# EPICS substitutions: apps/caenHvApp/Db/subs/HVECAL5_SPARES.substitutions
#
#This file was autogenerated by mkHVEpics.C on: Wed Nov  2 16:01:55 2016
#Substitutions for crate: HVECAL5 SPARES
#
file "db/caenhv.db" {
        pattern { Cr,    CrName,         CrType, Sl,     Ch,    Sys,     Det,    Element,                CScode, pwonoff, v0set,  i0set,   trip,    rampup,  rampdn, svmax,   enable}
		{"10",	"HVECAL5",	"4527",	"09",	"00",	"HV",	"HVECAL5",	"SPARE_Sl09_Ch00",	"#C2314", "S2816", "S512", "S1280", "S2560", "S1024", "S768", "S3328", "S256"}
		{"10",	"HVECAL5",	"4527",	"09",	"01",	"HV",	"HVECAL5",	"SPARE_Sl09_Ch01",	"#C2314", "S2817", "S513", "S1281", "S2561", "S1025", "S769", "S3329", "S257"}
		{"10",	"HVECAL5",	"4527",	"09",	"02",	"HV",	"HVECAL5",	"SPARE_Sl09_Ch02",	"#C2314", "S2818", "S514", "S1282", "S2562", "S1026", "S770", "S3330", "S258"}
		{"10",	"HVECAL5",	"4527",	"09",	"03",	"HV",	"HVECAL5",	"SPARE_Sl09_Ch03",	"#C2314", "S2819", "S515", "S1283", "S2563", "S1027", "S771", "S3331", "S259"}
		{"10",	"HVECAL5",	"4527",	"09",	"04",	"HV",	"HVECAL5",	"SPARE_Sl09_Ch04",	"#C2314", "S2820", "S516", "S1284", "S2564", "S1028", "S772", "S3332", "S260"}
		{"10",	"HVECAL5",	"4527",	"09",	"05",	"HV",	"HVECAL5",	"SPARE_Sl09_Ch05",	"#C2314", "S2821", "S517", "S1285", "S2565", "S1029", "S773", "S3333", "S261"}
		{"10",	"HVECAL5",	"4527",	"09",	"06",	"HV",	"HVECAL5",	"SPARE_Sl09_Ch06",	"#C2314", "S2822", "S518", "S1286", "S2566", "S1030", "S774", "S3334", "S262"}
		{"10",	"HVECAL5",	"4527",	"09",	"07",	"HV",	"HVECAL5",	"SPARE_Sl09_Ch07",	"#C2314", "S2823", "S519", "S1287", "S2567", "S1031", "S775", "S3335", "S263"}
		{"10",	"HVECAL5",	"4527",	"09",	"08",	"HV",	"HVECAL5",	"SPARE_Sl09_Ch08",	"#C2314", "S2824", "S520", "S1288", "S2568", "S1032", "S776", "S3336", "S264"}
		{"10",	"HVECAL5",	"4527",	"09",	"09",	"HV",	"HVECAL5",	"SPARE_Sl09_Ch09",	"#C2314", "S2825", "S521", "S1289", "S2569", "S1033", "S777", "S3337", "S265"}
		{"10",	"HVECAL5",	"4527",	"09",	"10",	"HV",	"HVECAL5",	"SPARE_Sl09_Ch10",	"#C2314", "S2826", "S522", "S1290", "S2570", "S1034", "S778", "S3338", "S266"}
		{"10",	"HVECAL5",	"4527",	"09",	"11",	"HV",	"HVECAL5",	"SPARE_Sl09_Ch11",	"#C2314", "S2827", "S523", "S1291", "S2571", "S1035", "S779", "S3339", "S267"}
		{"10",	"HVECAL5",	"4527",	"09",	"12",	"HV",	"HVECAL5",	"SPARE_Sl09_Ch12",	"#C2314", "S2828", "S524", "S1292", "S2572", "S1036", "S780", "S3340", "S268"}
		{"10",	"HVECAL5",	"4527",	"09",	"13",	"HV",	"HVECAL5",	"SPARE_Sl09_Ch13",	"#C2314", "S2829", "S525", "S1293", "S2573", "S1037", "S781", "S3341", "S269"}
		{"10",	"HVECAL5",	"4527",	"09",	"14",	"HV",	"HVECAL5",	"SPARE_Sl09_Ch14",	"#C2314", "S2830", "S526", "S1294", "S2574", "S1038", "S782", "S3342", "S270"}
		{"10",	"HVECAL5",	"4527",	"09",	"15",	"HV",	"HVECAL5",	"SPARE_Sl09_Ch15",	"#C2314", "S2831", "S527", "S1295", "S2575", "S1039", "S783", "S3343", "S271"}
		{"10",	"HVECAL5",	"4527",	"09",	"16",	"HV",	"HVECAL5",	"SPARE_Sl09_Ch16",	"#C2314", "S2832", "S528", "S1296", "S2576", "S1040", "S784", "S3344", "S272"}
		{"10",	"HVECAL5",	"4527",	"09",	"17",	"HV",	"HVECAL5",	"SPARE_Sl09_Ch17",	"#C2314", "S2833", "S529", "S1297", "S2577", "S1041", "S785", "S3345", "S273"}
		{"10",	"HVECAL5",	"4527",	"09",	"18",	"HV",	"HVECAL5",	"SPARE_Sl09_Ch18",	"#C2314", "S2834", "S530", "S1298", "S2578", "S1042", "S786", "S3346", "S274"}
		{"10",	"HVECAL5",	"4527",	"09",	"19",	"HV",	"HVECAL5",	"SPARE_Sl09_Ch19",	"#C2314", "S2835", "S531", "S1299", "S2579", "S1043", "S787", "S3347", "S275"}
		{"10",	"HVECAL5",	"4527",	"09",	"20",	"HV",	"HVECAL5",	"SPARE_Sl09_Ch20",	"#C2314", "S2836", "S532", "S1300", "S2580", "S1044", "S788", "S3348", "S276"}
		{"10",	"HVECAL5",	"4527",	"09",	"21",	"HV",	"HVECAL5",	"SPARE_Sl09_Ch21",	"#C2314", "S2837", "S533", "S1301", "S2581", "S1045", "S789", "S3349", "S277"}
		{"10",	"HVECAL5",	"4527",	"09",	"22",	"HV",	"HVECAL5",	"SPARE_Sl09_Ch22",	"#C2314", "S2838", "S534", "S1302", "S2582", "S1046", "S790", "S3350", "S278"}
		{"10",	"HVECAL5",	"4527",	"09",	"23",	"HV",	"HVECAL5",	"SPARE_Sl09_Ch23",	"#C2314", "S2839", "S535", "S1303", "S2583", "S1047", "S791", "S3351", "S279"}
		{"10",	"HVECAL5",	"4527",	"10",	"00",	"HV",	"HVECAL5",	"SPARE_Sl10_Ch00",	"#C2570", "S2816", "S512", "S1280", "S2560", "S1024", "S768", "S3328", "S256"}
		{"10",	"HVECAL5",	"4527",	"10",	"01",	"HV",	"HVECAL5",	"SPARE_Sl10_Ch01",	"#C2570", "S2817", "S513", "S1281", "S2561", "S1025", "S769", "S3329", "S257"}
		{"10",	"HVECAL5",	"4527",	"10",	"02",	"HV",	"HVECAL5",	"SPARE_Sl10_Ch02",	"#C2570", "S2818", "S514", "S1282", "S2562", "S1026", "S770", "S3330", "S258"}
		{"10",	"HVECAL5",	"4527",	"10",	"03",	"HV",	"HVECAL5",	"SPARE_Sl10_Ch03",	"#C2570", "S2819", "S515", "S1283", "S2563", "S1027", "S771", "S3331", "S259"}
		{"10",	"HVECAL5",	"4527",	"10",	"04",	"HV",	"HVECAL5",	"SPARE_Sl10_Ch04",	"#C2570", "S2820", "S516", "S1284", "S2564", "S1028", "S772", "S3332", "S260"}
		{"10",	"HVECAL5",	"4527",	"10",	"05",	"HV",	"HVECAL5",	"SPARE_Sl10_Ch05",	"#C2570", "S2821", "S517", "S1285", "S2565", "S1029", "S773", "S3333", "S261"}
		{"10",	"HVECAL5",	"4527",	"10",	"06",	"HV",	"HVECAL5",	"SPARE_Sl10_Ch06",	"#C2570", "S2822", "S518", "S1286", "S2566", "S1030", "S774", "S3334", "S262"}
		{"10",	"HVECAL5",	"4527",	"10",	"07",	"HV",	"HVECAL5",	"SPARE_Sl10_Ch07",	"#C2570", "S2823", "S519", "S1287", "S2567", "S1031", "S775", "S3335", "S263"}
		{"10",	"HVECAL5",	"4527",	"10",	"08",	"HV",	"HVECAL5",	"SPARE_Sl10_Ch08",	"#C2570", "S2824", "S520", "S1288", "S2568", "S1032", "S776", "S3336", "S264"}
		{"10",	"HVECAL5",	"4527",	"10",	"09",	"HV",	"HVECAL5",	"SPARE_Sl10_Ch09",	"#C2570", "S2825", "S521", "S1289", "S2569", "S1033", "S777", "S3337", "S265"}
		{"10",	"HVECAL5",	"4527",	"10",	"10",	"HV",	"HVECAL5",	"SPARE_Sl10_Ch10",	"#C2570", "S2826", "S522", "S1290", "S2570", "S1034", "S778", "S3338", "S266"}
		{"10",	"HVECAL5",	"4527",	"10",	"11",	"HV",	"HVECAL5",	"SPARE_Sl10_Ch11",	"#C2570", "S2827", "S523", "S1291", "S2571", "S1035", "S779", "S3339", "S267"}
		{"10",	"HVECAL5",	"4527",	"10",	"12",	"HV",	"HVECAL5",	"SPARE_Sl10_Ch12",	"#C2570", "S2828", "S524", "S1292", "S2572", "S1036", "S780", "S3340", "S268"}
		{"10",	"HVECAL5",	"4527",	"10",	"13",	"HV",	"HVECAL5",	"SPARE_Sl10_Ch13",	"#C2570", "S2829", "S525", "S1293", "S2573", "S1037", "S781", "S3341", "S269"}
		{"10",	"HVECAL5",	"4527",	"10",	"14",	"HV",	"HVECAL5",	"SPARE_Sl10_Ch14",	"#C2570", "S2830", "S526", "S1294", "S2574", "S1038", "S782", "S3342", "S270"}
		{"10",	"HVECAL5",	"4527",	"10",	"15",	"HV",	"HVECAL5",	"SPARE_Sl10_Ch15",	"#C2570", "S2831", "S527", "S1295", "S2575", "S1039", "S783", "S3343", "S271"}
		{"10",	"HVECAL5",	"4527",	"10",	"16",	"HV",	"HVECAL5",	"SPARE_Sl10_Ch16",	"#C2570", "S2832", "S528", "S1296", "S2576", "S1040", "S784", "S3344", "S272"}
		{"10",	"HVECAL5",	"4527",	"10",	"17",	"HV",	"HVECAL5",	"SPARE_Sl10_Ch17",	"#C2570", "S2833", "S529", "S1297", "S2577", "S1041", "S785", "S3345", "S273"}
		{"10",	"HVECAL5",	"4527",	"10",	"18",	"HV",	"HVECAL5",	"SPARE_Sl10_Ch18",	"#C2570", "S2834", "S530", "S1298", "S2578", "S1042", "S786", "S3346", "S274"}
		{"10",	"HVECAL5",	"4527",	"10",	"19",	"HV",	"HVECAL5",	"SPARE_Sl10_Ch19",	"#C2570", "S2835", "S531", "S1299", "S2579", "S1043", "S787", "S3347", "S275"}
		{"10",	"HVECAL5",	"4527",	"10",	"20",	"HV",	"HVECAL5",	"SPARE_Sl10_Ch20",	"#C2570", "S2836", "S532", "S1300", "S2580", "S1044", "S788", "S3348", "S276"}
		{"10",	"HVECAL5",	"4527",	"10",	"21",	"HV",	"HVECAL5",	"SPARE_Sl10_Ch21",	"#C2570", "S2837", "S533", "S1301", "S2581", "S1045", "S789", "S3349", "S277"}
		{"10",	"HVECAL5",	"4527",	"10",	"22",	"HV",	"HVECAL5",	"SPARE_Sl10_Ch22",	"#C2570", "S2838", "S534", "S1302", "S2582", "S1046", "S790", "S3350", "S278"}
		{"10",	"HVECAL5",	"4527",	"10",	"23",	"HV",	"HVECAL5",	"SPARE_Sl10_Ch23",	"#C2570", "S2839", "S535", "S1303", "S2583", "S1047", "S791", "S3351", "S279"}
		{"10",	"HVECAL5",	"4527",	"11",	"00",	"HV",	"HVECAL5",	"SPARE_Sl11_Ch00",	"#C2826", "S2816", "S512", "S1280", "S2560", "S1024", "S768", "S3328", "S256"}
		{"10",	"HVECAL5",	"4527",	"11",	"01",	"HV",	"HVECAL5",	"SPARE_Sl11_Ch01",	"#C2826", "S2817", "S513", "S1281", "S2561", "S1025", "S769", "S3329", "S257"}
		{"10",	"HVECAL5",	"4527",	"11",	"02",	"HV",	"HVECAL5",	"SPARE_Sl11_Ch02",	"#C2826", "S2818", "S514", "S1282", "S2562", "S1026", "S770", "S3330", "S258"}
		{"10",	"HVECAL5",	"4527",	"11",	"03",	"HV",	"HVECAL5",	"SPARE_Sl11_Ch03",	"#C2826", "S2819", "S515", "S1283", "S2563", "S1027", "S771", "S3331", "S259"}
		{"10",	"HVECAL5",	"4527",	"11",	"04",	"HV",	"HVECAL5",	"SPARE_Sl11_Ch04",	"#C2826", "S2820", "S516", "S1284", "S2564", "S1028", "S772", "S3332", "S260"}
		{"10",	"HVECAL5",	"4527",	"11",	"05",	"HV",	"HVECAL5",	"SPARE_Sl11_Ch05",	"#C2826", "S2821", "S517", "S1285", "S2565", "S1029", "S773", "S3333", "S261"}
		{"10",	"HVECAL5",	"4527",	"11",	"06",	"HV",	"HVECAL5",	"SPARE_Sl11_Ch06",	"#C2826", "S2822", "S518", "S1286", "S2566", "S1030", "S774", "S3334", "S262"}
		{"10",	"HVECAL5",	"4527",	"11",	"07",	"HV",	"HVECAL5",	"SPARE_Sl11_Ch07",	"#C2826", "S2823", "S519", "S1287", "S2567", "S1031", "S775", "S3335", "S263"}
		{"10",	"HVECAL5",	"4527",	"11",	"08",	"HV",	"HVECAL5",	"SPARE_Sl11_Ch08",	"#C2826", "S2824", "S520", "S1288", "S2568", "S1032", "S776", "S3336", "S264"}
		{"10",	"HVECAL5",	"4527",	"11",	"09",	"HV",	"HVECAL5",	"SPARE_Sl11_Ch09",	"#C2826", "S2825", "S521", "S1289", "S2569", "S1033", "S777", "S3337", "S265"}
		{"10",	"HVECAL5",	"4527",	"11",	"10",	"HV",	"HVECAL5",	"SPARE_Sl11_Ch10",	"#C2826", "S2826", "S522", "S1290", "S2570", "S1034", "S778", "S3338", "S266"}
		{"10",	"HVECAL5",	"4527",	"11",	"11",	"HV",	"HVECAL5",	"SPARE_Sl11_Ch11",	"#C2826", "S2827", "S523", "S1291", "S2571", "S1035", "S779", "S3339", "S267"}
		{"10",	"HVECAL5",	"4527",	"11",	"12",	"HV",	"HVECAL5",	"SPARE_Sl11_Ch12",	"#C2826", "S2828", "S524", "S1292", "S2572", "S1036", "S780", "S3340", "S268"}
		{"10",	"HVECAL5",	"4527",	"11",	"13",	"HV",	"HVECAL5",	"SPARE_Sl11_Ch13",	"#C2826", "S2829", "S525", "S1293", "S2573", "S1037", "S781", "S3341", "S269"}
		{"10",	"HVECAL5",	"4527",	"11",	"14",	"HV",	"HVECAL5",	"SPARE_Sl11_Ch14",	"#C2826", "S2830", "S526", "S1294", "S2574", "S1038", "S782", "S3342", "S270"}
		{"10",	"HVECAL5",	"4527",	"11",	"15",	"HV",	"HVECAL5",	"SPARE_Sl11_Ch15",	"#C2826", "S2831", "S527", "S1295", "S2575", "S1039", "S783", "S3343", "S271"}
		{"10",	"HVECAL5",	"4527",	"11",	"16",	"HV",	"HVECAL5",	"SPARE_Sl11_Ch16",	"#C2826", "S2832", "S528", "S1296", "S2576", "S1040", "S784", "S3344", "S272"}
		{"10",	"HVECAL5",	"4527",	"11",	"17",	"HV",	"HVECAL5",	"SPARE_Sl11_Ch17",	"#C2826", "S2833", "S529", "S1297", "S2577", "S1041", "S785", "S3345", "S273"}
		{"10",	"HVECAL5",	"4527",	"11",	"18",	"HV",	"HVECAL5",	"SPARE_Sl11_Ch18",	"#C2826", "S2834", "S530", "S1298", "S2578", "S1042", "S786", "S3346", "S274"}
		{"10",	"HVECAL5",	"4527",	"11",	"19",	"HV",	"HVECAL5",	"SPARE_Sl11_Ch19",	"#C2826", "S2835", "S531", "S1299", "S2579", "S1043", "S787", "S3347", "S275"}
		{"10",	"HVECAL5",	"4527",	"11",	"20",	"HV",	"HVECAL5",	"SPARE_Sl11_Ch20",	"#C2826", "S2836", "S532", "S1300", "S2580", "S1044", "S788", "S3348", "S276"}
		{"10",	"HVECAL5",	"4527",	"11",	"21",	"HV",	"HVECAL5",	"SPARE_Sl11_Ch21",	"#C2826", "S2837", "S533", "S1301", "S2581", "S1045", "S789", "S3349", "S277"}
		{"10",	"HVECAL5",	"4527",	"11",	"22",	"HV",	"HVECAL5",	"SPARE_Sl11_Ch22",	"#C2826", "S2838", "S534", "S1302", "S2582", "S1046", "S790", "S3350", "S278"}
		{"10",	"HVECAL5",	"4527",	"11",	"23",	"HV",	"HVECAL5",	"SPARE_Sl11_Ch23",	"#C2826", "S2839", "S535", "S1303", "S2583", "S1047", "S791", "S3351", "S279"}
		{"10",	"HVECAL5",	"4527",	"12",	"00",	"HV",	"HVECAL5",	"SPARE_Sl12_Ch00",	"#C3082", "S2816", "S512", "S1280", "S2560", "S1024", "S768", "S3328", "S256"}
		{"10",	"HVECAL5",	"4527",	"12",	"01",	"HV",	"HVECAL5",	"SPARE_Sl12_Ch01",	"#C3082", "S2817", "S513", "S1281", "S2561", "S1025", "S769", "S3329", "S257"}
		{"10",	"HVECAL5",	"4527",	"12",	"02",	"HV",	"HVECAL5",	"SPARE_Sl12_Ch02",	"#C3082", "S2818", "S514", "S1282", "S2562", "S1026", "S770", "S3330", "S258"}
		{"10",	"HVECAL5",	"4527",	"12",	"03",	"HV",	"HVECAL5",	"SPARE_Sl12_Ch03",	"#C3082", "S2819", "S515", "S1283", "S2563", "S1027", "S771", "S3331", "S259"}
		{"10",	"HVECAL5",	"4527",	"12",	"04",	"HV",	"HVECAL5",	"SPARE_Sl12_Ch04",	"#C3082", "S2820", "S516", "S1284", "S2564", "S1028", "S772", "S3332", "S260"}
		{"10",	"HVECAL5",	"4527",	"12",	"05",	"HV",	"HVECAL5",	"SPARE_Sl12_Ch05",	"#C3082", "S2821", "S517", "S1285", "S2565", "S1029", "S773", "S3333", "S261"}
		{"10",	"HVECAL5",	"4527",	"12",	"06",	"HV",	"HVECAL5",	"SPARE_Sl12_Ch06",	"#C3082", "S2822", "S518", "S1286", "S2566", "S1030", "S774", "S3334", "S262"}
		{"10",	"HVECAL5",	"4527",	"12",	"07",	"HV",	"HVECAL5",	"SPARE_Sl12_Ch07",	"#C3082", "S2823", "S519", "S1287", "S2567", "S1031", "S775", "S3335", "S263"}
		{"10",	"HVECAL5",	"4527",	"12",	"08",	"HV",	"HVECAL5",	"SPARE_Sl12_Ch08",	"#C3082", "S2824", "S520", "S1288", "S2568", "S1032", "S776", "S3336", "S264"}
		{"10",	"HVECAL5",	"4527",	"12",	"09",	"HV",	"HVECAL5",	"SPARE_Sl12_Ch09",	"#C3082", "S2825", "S521", "S1289", "S2569", "S1033", "S777", "S3337", "S265"}
		{"10",	"HVECAL5",	"4527",	"12",	"10",	"HV",	"HVECAL5",	"SPARE_Sl12_Ch10",	"#C3082", "S2826", "S522", "S1290", "S2570", "S1034", "S778", "S3338", "S266"}
		{"10",	"HVECAL5",	"4527",	"12",	"11",	"HV",	"HVECAL5",	"SPARE_Sl12_Ch11",	"#C3082", "S2827", "S523", "S1291", "S2571", "S1035", "S779", "S3339", "S267"}
		{"10",	"HVECAL5",	"4527",	"12",	"12",	"HV",	"HVECAL5",	"SPARE_Sl12_Ch12",	"#C3082", "S2828", "S524", "S1292", "S2572", "S1036", "S780", "S3340", "S268"}
		{"10",	"HVECAL5",	"4527",	"12",	"13",	"HV",	"HVECAL5",	"SPARE_Sl12_Ch13",	"#C3082", "S2829", "S525", "S1293", "S2573", "S1037", "S781", "S3341", "S269"}
		{"10",	"HVECAL5",	"4527",	"12",	"14",	"HV",	"HVECAL5",	"SPARE_Sl12_Ch14",	"#C3082", "S2830", "S526", "S1294", "S2574", "S1038", "S782", "S3342", "S270"}
		{"10",	"HVECAL5",	"4527",	"12",	"15",	"HV",	"HVECAL5",	"SPARE_Sl12_Ch15",	"#C3082", "S2831", "S527", "S1295", "S2575", "S1039", "S783", "S3343", "S271"}
		{"10",	"HVECAL5",	"4527",	"12",	"16",	"HV",	"HVECAL5",	"SPARE_Sl12_Ch16",	"#C3082", "S2832", "S528", "S1296", "S2576", "S1040", "S784", "S3344", "S272"}
		{"10",	"HVECAL5",	"4527",	"12",	"17",	"HV",	"HVECAL5",	"SPARE_Sl12_Ch17",	"#C3082", "S2833", "S529", "S1297", "S2577", "S1041", "S785", "S3345", "S273"}
		{"10",	"HVECAL5",	"4527",	"12",	"18",	"HV",	"HVECAL5",	"SPARE_Sl12_Ch18",	"#C3082", "S2834", "S530", "S1298", "S2578", "S1042", "S786", "S3346", "S274"}
		{"10",	"HVECAL5",	"4527",	"12",	"19",	"HV",	"HVECAL5",	"SPARE_Sl12_Ch19",	"#C3082", "S2835", "S531", "S1299", "S2579", "S1043", "S787", "S3347", "S275"}
		{"10",	"HVECAL5",	"4527",	"12",	"20",	"HV",	"HVECAL5",	"SPARE_Sl12_Ch20",	"#C3082", "S2836", "S532", "S1300", "S2580", "S1044", "S788", "S3348", "S276"}
		{"10",	"HVECAL5",	"4527",	"12",	"21",	"HV",	"HVECAL5",	"SPARE_Sl12_Ch21",	"#C3082", "S2837", "S533", "S1301", "S2581", "S1045", "S789", "S3349", "S277"}
		{"10",	"HVECAL5",	"4527",	"12",	"22",	"HV",	"HVECAL5",	"SPARE_Sl12_Ch22",	"#C3082", "S2838", "S534", "S1302", "S2582", "S1046", "S790", "S3350", "S278"}
		{"10",	"HVECAL5",	"4527",	"12",	"23",	"HV",	"HVECAL5",	"SPARE_Sl12_Ch23",	"#C3082", "S2839", "S535", "S1303", "S2583", "S1047", "S791", "S3351", "S279"}
		{"10",	"HVECAL5",	"4527",	"13",	"00",	"HV",	"HVECAL5",	"SPARE_Sl13_Ch00",	"#C3338", "S2816", "S512", "S1280", "S2560", "S1024", "S768", "S3328", "S256"}
		{"10",	"HVECAL5",	"4527",	"13",	"01",	"HV",	"HVECAL5",	"SPARE_Sl13_Ch01",	"#C3338", "S2817", "S513", "S1281", "S2561", "S1025", "S769", "S3329", "S257"}
		{"10",	"HVECAL5",	"4527",	"13",	"02",	"HV",	"HVECAL5",	"SPARE_Sl13_Ch02",	"#C3338", "S2818", "S514", "S1282", "S2562", "S1026", "S770", "S3330", "S258"}
		{"10",	"HVECAL5",	"4527",	"13",	"03",	"HV",	"HVECAL5",	"SPARE_Sl13_Ch03",	"#C3338", "S2819", "S515", "S1283", "S2563", "S1027", "S771", "S3331", "S259"}
		{"10",	"HVECAL5",	"4527",	"13",	"04",	"HV",	"HVECAL5",	"SPARE_Sl13_Ch04",	"#C3338", "S2820", "S516", "S1284", "S2564", "S1028", "S772", "S3332", "S260"}
		{"10",	"HVECAL5",	"4527",	"13",	"05",	"HV",	"HVECAL5",	"SPARE_Sl13_Ch05",	"#C3338", "S2821", "S517", "S1285", "S2565", "S1029", "S773", "S3333", "S261"}
		{"10",	"HVECAL5",	"4527",	"13",	"06",	"HV",	"HVECAL5",	"SPARE_Sl13_Ch06",	"#C3338", "S2822", "S518", "S1286", "S2566", "S1030", "S774", "S3334", "S262"}
		{"10",	"HVECAL5",	"4527",	"13",	"07",	"HV",	"HVECAL5",	"SPARE_Sl13_Ch07",	"#C3338", "S2823", "S519", "S1287", "S2567", "S1031", "S775", "S3335", "S263"}
		{"10",	"HVECAL5",	"4527",	"13",	"08",	"HV",	"HVECAL5",	"SPARE_Sl13_Ch08",	"#C3338", "S2824", "S520", "S1288", "S2568", "S1032", "S776", "S3336", "S264"}
		{"10",	"HVECAL5",	"4527",	"13",	"09",	"HV",	"HVECAL5",	"SPARE_Sl13_Ch09",	"#C3338", "S2825", "S521", "S1289", "S2569", "S1033", "S777", "S3337", "S265"}
		{"10",	"HVECAL5",	"4527",	"13",	"10",	"HV",	"HVECAL5",	"SPARE_Sl13_Ch10",	"#C3338", "S2826", "S522", "S1290", "S2570", "S1034", "S778", "S3338", "S266"}
		{"10",	"HVECAL5",	"4527",	"13",	"11",	"HV",	"HVECAL5",	"SPARE_Sl13_Ch11",	"#C3338", "S2827", "S523", "S1291", "S2571", "S1035", "S779", "S3339", "S267"}
		{"10",	"HVECAL5",	"4527",	"13",	"12",	"HV",	"HVECAL5",	"SPARE_Sl13_Ch12",	"#C3338", "S2828", "S524", "S1292", "S2572", "S1036", "S780", "S3340", "S268"}
		{"10",	"HVECAL5",	"4527",	"13",	"13",	"HV",	"HVECAL5",	"SPARE_Sl13_Ch13",	"#C3338", "S2829", "S525", "S1293", "S2573", "S1037", "S781", "S3341", "S269"}
		{"10",	"HVECAL5",	"4527",	"13",	"14",	"HV",	"HVECAL5",	"SPARE_Sl13_Ch14",	"#C3338", "S2830", "S526", "S1294", "S2574", "S1038", "S782", "S3342", "S270"}
		{"10",	"HVECAL5",	"4527",	"13",	"15",	"HV",	"HVECAL5",	"SPARE_Sl13_Ch15",	"#C3338", "S2831", "S527", "S1295", "S2575", "S1039", "S783", "S3343", "S271"}
		{"10",	"HVECAL5",	"4527",	"13",	"16",	"HV",	"HVECAL5",	"SPARE_Sl13_Ch16",	"#C3338", "S2832", "S528", "S1296", "S2576", "S1040", "S784", "S3344", "S272"}
		{"10",	"HVECAL5",	"4527",	"13",	"17",	"HV",	"HVECAL5",	"SPARE_Sl13_Ch17",	"#C3338", "S2833", "S529", "S1297", "S2577", "S1041", "S785", "S3345", "S273"}
		{"10",	"HVECAL5",	"4527",	"13",	"18",	"HV",	"HVECAL5",	"SPARE_Sl13_Ch18",	"#C3338", "S2834", "S530", "S1298", "S2578", "S1042", "S786", "S3346", "S274"}
		{"10",	"HVECAL5",	"4527",	"13",	"19",	"HV",	"HVECAL5",	"SPARE_Sl13_Ch19",	"#C3338", "S2835", "S531", "S1299", "S2579", "S1043", "S787", "S3347", "S275"}
		{"10",	"HVECAL5",	"4527",	"13",	"20",	"HV",	"HVECAL5",	"SPARE_Sl13_Ch20",	"#C3338", "S2836", "S532", "S1300", "S2580", "S1044", "S788", "S3348", "S276"}
		{"10",	"HVECAL5",	"4527",	"13",	"21",	"HV",	"HVECAL5",	"SPARE_Sl13_Ch21",	"#C3338", "S2837", "S533", "S1301", "S2581", "S1045", "S789", "S3349", "S277"}
		{"10",	"HVECAL5",	"4527",	"13",	"22",	"HV",	"HVECAL5",	"SPARE_Sl13_Ch22",	"#C3338", "S2838", "S534", "S1302", "S2582", "S1046", "S790", "S3350", "S278"}
		{"10",	"HVECAL5",	"4527",	"13",	"23",	"HV",	"HVECAL5",	"SPARE_Sl13_Ch23",	"#C3338", "S2839", "S535", "S1303", "S2583", "S1047", "S791", "S3351", "S279"}
		{"10",	"HVECAL5",	"4527",	"14",	"18",	"HV",	"HVECAL5",	"SPARE_Sl14_Ch18",	"#C3594", "S2834", "S530", "S1298", "S2578", "S1042", "S786", "S3346", "S274"}
		{"10",	"HVECAL5",	"4527",	"14",	"19",	"HV",	"HVECAL5",	"SPARE_Sl14_Ch19",	"#C3594", "S2835", "S531", "S1299", "S2579", "S1043", "S787", "S3347", "S275"}
		{"10",	"HVECAL5",	"4527",	"14",	"20",	"HV",	"HVECAL5",	"SPARE_Sl14_Ch20",	"#C3594", "S2836", "S532", "S1300", "S2580", "S1044", "S788", "S3348", "S276"}
		{"10",	"HVECAL5",	"4527",	"14",	"21",	"HV",	"HVECAL5",	"SPARE_Sl14_Ch21",	"#C3594", "S2837", "S533", "S1301", "S2581", "S1045", "S789", "S3349", "S277"}
		{"10",	"HVECAL5",	"4527",	"14",	"22",	"HV",	"HVECAL5",	"SPARE_Sl14_Ch22",	"#C3594", "S2838", "S534", "S1302", "S2582", "S1046", "S790", "S3350", "S278"}
		{"10",	"HVECAL5",	"4527",	"14",	"23",	"HV",	"HVECAL5",	"SPARE_Sl14_Ch23",	"#C3594", "S2839", "S535", "S1303", "S2583", "S1047", "S791", "S3351", "S279"}
		{"10",	"HVECAL5",	"4527",	"15",	"18",	"HV",	"HVECAL5",	"SPARE_Sl15_Ch18",	"#C3850", "S2834", "S530", "S1298", "S2578", "S1042", "S786", "S3346", "S274"}
		{"10",	"HVECAL5",	"4527",	"15",	"19",	"HV",	"HVECAL5",	"SPARE_Sl15_Ch19",	"#C3850", "S2835", "S531", "S1299", "S2579", "S1043", "S787", "S3347", "S275"}
		{"10",	"HVECAL5",	"4527",	"15",	"20",	"HV",	"HVECAL5",	"SPARE_Sl15_Ch20",	"#C3850", "S2836", "S532", "S1300", "S2580", "S1044", "S788", "S3348", "S276"}
		{"10",	"HVECAL5",	"4527",	"15",	"21",	"HV",	"HVECAL5",	"SPARE_Sl15_Ch21",	"#C3850", "S2837", "S533", "S1301", "S2581", "S1045", "S789", "S3349", "S277"}
		{"10",	"HVECAL5",	"4527",	"15",	"22",	"HV",	"HVECAL5",	"SPARE_Sl15_Ch22",	"#C3850", "S2838", "S534", "S1302", "S2582", "S1046", "S790", "S3350", "S278"}
		{"10",	"HVECAL5",	"4527",	"15",	"23",	"HV",	"HVECAL5",	"SPARE_Sl15_Ch23",	"#C3850", "S2839", "S535", "S1303", "S2583", "S1047", "S791", "S3351", "S279"}
}
